TEXTLIST TL_GroupState
  0 = 'UNKNOWN'
  1 = 'RUN'
  2 = 'STOP'
  3 = 'SAFE'
  4 = 'ERROR'
  5 = 'RESET'
   = ''
END_TEXTLIST

(* stored: Version 1.1.0.1, ProductVersion 3.1.4022.12
   TextList TL_GroupState: Id {9df8e400-d8ab-4794-8d65-2fbe073d1992} *)
